FUNCTION "FC_Local_Class_Dir_T_this_is_a_pretty_long_title" : Void
TITLE = %version: 5.09 % %Commit:  c3808b61 % CN: 33
{ S7_Optimized_Access := 'FALSE' }
FAMILY : Tubtrax
VERSION : 0.0
//Function:
//Retreive preferred direction for instance DB and check the local constrains
//local constrains are SBT and OBT Class
//
//
//SOURCE
//%Project:      allcttt %
//%Repo:         a_ttt %
//%Commit:       c3808b61 %
//%DateTimeUTC:  2023-12-11T14:59:55 %
//
//%HISTORY%
//Issue:        Commit:  Date:      Version: Author:              Description:
//------------- -------- ---------- -------- -------------------- ------------------------------------------------------------------------------
//ALLCTTT-4059  c3808b61 2023-12-11 5.09     Pascal van Kempen    Added history table
//ALLCTTT-4042  a864e0dd 2023-12-06 5.08     Harm Hopmans         Renamed folders that contained space character
//ALLCTTT-4042  55fd833f 2023-12-05 5.07     Henri de Leijer      First step to remove the library files
//ALLCTTT-272   544e4e84 2020-12-10 5.06     Pascal van Kempen    removed keywords
//ALLCTTT-272   9d531fbf 2020-12-10 5.05     Pascal van Kempen    Revert corrected checkin sequence for determining version information properly
//ALLCTTT-272   ae3fa862 2020-12-10 5.04     Pascal van Kempen    corrected checkin sequence for determining version information properly
//ALLCTTT-272   5a1edb78 2020-12-10 5.03     Pascal van Kempen    Revert keywords updates
//ALLCTTT-272   8d62c219 2020-12-10 5.02     Pascal van Kempen    keywords updates
//ALLCTTT-272   31a64871 2020-12-10 5.01     Pascal van Kempen    initial import
//
//Modification History:                                 By:      Date:     Rev:
//----------------------------------------------------  -------  --------  -----
//mco#3663: Updated Pointer address                     inragr   06-07-20   2.02
//ra#31964: Based on 2.15.0.0 version 1.02              nlhhop   14-01-19   2.01
//
//Description:
//Retreive preferred direction for instance DB and check the local constrains
//local constrains are SBT and OBT Class
   VAR_INPUT
      i_Class_SBT : Bool;   // When TRUE tub class is SBT
      i_Class_OBT : Bool;   // When TRUE tub class is OBT
      i_ANY_Preferred_Dir : Any;   // ANY pointer to the preferred direction
      i_CFG_Local_SBT_Dir : Int;   // CFG: Local Direction for SBTs. Direction 1 or 2 or 'don't care'(0)
      i_CFG_Local_OBT_Dir : Int;   // CFG: Local Direction for OBTs. Direction 1 or 2 or 'don't care'(0)
      i_DINO : Int;   // DI number of instance used
   END_VAR

   VAR_TEMP
      t_Destination : Int;   // Destination
      t_Preference_A : Byte;   // Preference for Direction A
      t_Preference_B : Byte;   // Preference for Direction B
      t_DecisionLvl : Byte;   // Decision Level
      t_FailedReason_A : Byte;   // Failed Reason for Direction A
      t_FailedReason_B : Byte;   // Failed Reason for Direction B
      t_Direction : Byte;   // Direction selected
      t_DINO : Int;   // DB number of instance
   END_VAR


BEGIN

END_FUNCTION

